PROGRAM P_Demo_UInt64Cmp64
VAR
    uliBatchA : T_ULARGE_INTEGER;; // A 线产量
    uliBatchB : T_ULARGE_INTEGER;; // B 线产量
    diResult  : DINT;; // 比较结果
    bCompare  : BOOL;; // 触发比较
END_VAR

// ============================================================
// Tc2_Utilities.UInt64Cmp64 演示程序（FUNCTION，单周期触发）
// ============================================================
// 场景：把两个生产批次的产量计数器排序，决定哪条线产量更高。
// 价值：替代手写两次 DWORD 比较 + 嵌套 IF；一次调用 + DINT 比较一目了然。
// 验证步骤：
//   1. 把本 PROGRAM 加到 PlcTask 调用列表
//   2. 编译 + 登录
//   3. 在线把 b... 触发位置 TRUE 一个周期
//   4. 观察输出变量是否符合期望
// ============================================================

IF bCompare THEN
    // -1: A 少 / 0: 持平 / 1: A 多
    diResult := UInt64Cmp64(uliBatchA, uliBatchB);
    bCompare := FALSE;
END_IF;

END_PROGRAM

(* stored: Version 1.1.0.1, ProductVersion 3.1.4024.5
   POU P_Demo_UInt64Cmp64: Id {fa112a32-9abe-5664-a145-2082506513be}, SpecialFunc None *)
